{attribute 'GeneratedUsingTerminal: ELX1058-0000-0016'}
{attribute addProperty BoxType "ELX1058-0000-0016"}
{attribute addProperty Id "Channel_1AT %I*Channel_31CEFA7F2Channel_2AT %I*Channel_31CEFA7F2Channel_3AT %I*Channel_31CEFA7F2Channel_4AT %I*Channel_31CEFA7F2Channel_5AT %I*Channel_31CEFA7F2Channel_6AT %I*Channel_31CEFA7F2Channel_7AT %I*Channel_31CEFA7F2Channel_8AT %I*Channel_31CEFA7F2WcStateAT %I*WcState_9091E0EB2InfoDataAT %I*InfoData_94A18F5E2"}
{attribute addProperty CRC "3336984425"}
{attribute addProperty Size "20"}
TYPE ELX1058_C6E65769 EXTENDS EtcSlaveTerminalBase_947E5A46 :
STRUCT
	{attribute addProperty Name "Channel_1"}
	Channel_1 : Channel_31CEFA7F;
	{attribute addProperty Name "Channel_2"}
	Channel_2 : Channel_31CEFA7F;
	{attribute addProperty Name "Channel_3"}
	Channel_3 : Channel_31CEFA7F;
	{attribute addProperty Name "Channel_4"}
	Channel_4 : Channel_31CEFA7F;
	{attribute addProperty Name "Channel_5"}
	Channel_5 : Channel_31CEFA7F;
	{attribute addProperty Name "Channel_6"}
	Channel_6 : Channel_31CEFA7F;
	{attribute addProperty Name "Channel_7"}
	Channel_7 : Channel_31CEFA7F;
	{attribute addProperty Name "Channel_8"}
	Channel_8 : Channel_31CEFA7F;
	{attribute addProperty Name "WcState"}
	WcState : WcState_9091E0EB;
	{attribute addProperty Name "InfoData"}
	InfoData : InfoData_94A18F5E;
END_STRUCT
END_TYPE

(* stored: Version 1.2.0.0, ProductVersion 3.1.4024.9
   DUT ELX1058_C6E65769: Id {7b23a402-c427-4513-86c2-b60d06e23598} *)
